// Usage:
// Call instance every scan while waiting for operations to complete.
// SetFileParams() Set the File directory 
// GetFile() Get the File.
// #various props: Observe the properties to see whether it passed the file checks.
// NextRow()
FUNCTION_BLOCK T_TxtFileWriter
VAR
// state vars.
	filePath : Tc2_Utilities.T_MaxString; // filepath
	
// backing properties	
	_Row : UINT; // current Row number (zero indexed)
	_Error : BOOL;
	_ErrorId : UDINT; // E_AdsErr
	
// Objects	
	fileWrite : T_FileWriteBase;(* Writes one record (line) *)
	
END_VAR

fileWrite();

{attribute 'monitoring' := 'call'}
// write buffer is empty
PROPERTY PUBLIC BufferClear : BOOL
GET
BufferClear := fileWrite.BufferClear;
END_GET
END_PROPERTY

{attribute 'monitoring' := 'call'}
// file operation in progress
PROPERTY PUBLIC Busy : BOOL
GET
Busy := fileWrite.Busy;
END_GET
END_PROPERTY

// Clears the buffer (does not write to file first).
METHOD PUBLIC ClearBuffer : BOOL
ClearBuffer := fileWrite.ClearWriteBuffer();
_Error := fileWrite.Error;
_ErrorId := fileWrite.ErrorId;

_Row := 0;
END_METHOD

{attribute 'monitoring' := 'call'}
// file oepration complete
PROPERTY PUBLIC Done : BOOL
GET
Done := fileWrite.Done;
END_GET
END_PROPERTY

{attribute 'monitoring' := 'call'}
// error with buffer or file operation
PROPERTY PUBLIC Error : BOOL
GET
Error := _Error := fileWrite.Error;
END_GET
END_PROPERTY

{attribute 'monitoring' := 'call'}
// error ID
PROPERTY PUBLIC ErrorId : UDINT
GET
ErrorId := _ErrorId := fileWrite.ErrorId;
END_GET
END_PROPERTY

// Add CRLF.
METHOD PUBLIC NewLine 
VAR_INST
	tempByte : BYTE;
END_VAR
VAR CONSTANT
	CARRIAGE_RETURN : BYTE := 16#D;
	LINE_FEED : BYTE := 16#A;
END_VAR
// load up CR.
tempByte := CARRIAGE_RETURN;

//Write.
fileWrite.AppendToBuffer(
		pDataForBuffer := ADR(tempByte),
		DataLength := SIZEOF(tempByte)
	);

// check for errors
IF Error THEN // Error looks at FileWrite.Error
	RETURN;
END_IF

// load up LF.
tempByte := LINE_FEED;

//Write.
fileWrite.AppendToBuffer(
		pDataForBuffer := ADR(tempByte),
		DataLength := SIZEOF(tempByte)
	);	

// check for errors
IF Error THEN // Error looks at FileWrite.Error
	RETURN;
END_IF

_Row := _Row + 1;
END_METHOD

// current row / line number
PROPERTY PUBLIC Row : UINT
GET
Row := _Row;
END_GET
END_PROPERTY

METHOD SetFileOpenMode
VAR_INPUT
	Append : BOOL;  // TRUE = append, FALSE = new
END_VAR
fileWrite.SetFileOpenMode( 
	Append := Append
);
END_METHOD

// Set the fully scoped file path *i.e. C:/Users/TwinCAT_User/MyText.txt
METHOD PUBLIC SetFileParams
VAR_INPUT
	FilePath : Tc2_Utilities.T_MaxString;
END_VAR
THIS^.filePath := FilePath; // for debug only.

fileWrite.SetFilePath(FilePath := FilePath);
END_METHOD

// Append string to current line
METHOD PUBLIC Write
VAR_INPUT
	Entry : TxtFileString; 
END_VAR

VAR_INST
	locStr : TxtFileString; // This has a valid memory address (inputs dont)
END_VAR
locStr := Entry;

// Add string.
fileWrite.AppendToBuffer(
	pDataForBuffer := ADR(locStr),
	DataLength := INT_TO_UDINT(LEN(locStr))
);

IF Error THEN // Error looks at FileWrite.Error
	RETURN;
END_IF
END_METHOD

// Append string to current line and add CRLF
METHOD PUBLIC WriteLine
VAR_INPUT
	Entry : TxtFileString; 
END_VAR
Write( Entry );
NewLine();
END_METHOD

// Write Buffer to File.
METHOD PUBLIC WriteToFile
IF Error THEN // Error looks at FileWrite.Error
	RETURN;
END_IF

fileWrite.StartWrite();
END_METHOD

END_FUNCTION_BLOCK

(* stored: Version 1.1.0.1, ProductVersion 3.1.4022.18
   POU T_TxtFileWriter: Id {7877d6c4-ac8f-4f51-9d97-6af63fe863ea}, SpecialFunc None
   Folder Methods: Id {557beb1e-a5df-4c97-b5bc-93adb3602a98}
   Folder Properties: Id {a117d6a1-550f-4f02-b9c4-485c0f0e05a4}
   Property BufferClear: Id {0522faa3-edb1-481d-acb2-0f2b11e4cfe4}
   Get Get: Id {f9d762fb-38dd-41b2-96e0-c0bd6fde12bc}
   Property Busy: Id {98647035-9385-4ef7-b495-16d35f24cc0f}
   Get Get: Id {515a2227-6b90-4704-800e-a8058a3dfea2}
   Method ClearBuffer: Id {126c2a98-1f93-4800-953b-913f8017ebdf}
   Property Done: Id {8806e327-c12a-45d4-9890-e2566aebb370}
   Get Get: Id {c0a2169e-6f0b-4f6f-b365-9e63bd56e566}
   Property Error: Id {4ae623c8-15ab-4af6-8d4e-41659dfa894b}
   Get Get: Id {ebfc107a-9475-4fd4-80d7-f90cc2a4cd9b}
   Property ErrorId: Id {45803805-22fb-411d-b0e9-216b3c32d09d}
   Get Get: Id {0a9283c3-c71d-4a18-a2e8-7748a5cb78b5}
   Method NewLine: Id {3fd784f3-5259-4473-a47f-b28775c734a6}
   Property Row: Id {0b28ec25-4b0f-46d2-9ab4-0723147d7906}
   Get Get: Id {4d37301a-2b10-4254-b922-02a3a36abbbd}
   Method SetFileOpenMode: Id {1153eed4-a1d5-05ce-3b75-e636b5cbc4f1}
   Method SetFileParams: Id {78577382-50fd-4e7d-96af-2c5f86f38a31}
   Method Write: Id {353e5bc5-048f-4831-8685-df85998479ca}
   Method WriteLine: Id {3bc6e7f9-ad51-4130-8a49-7cbd01169802}
   Method WriteToFile: Id {0024c296-5625-42b9-ae4c-00e67d013509} *)
